INTERFACE ITF_Heatpump EXTENDS ITF_StandardFB

PROPERTY HeatpumpState : eHeatpumpState
GET
END_GET
END_PROPERTY

PROPERTY OperationMode : eHeatpumpMode
SET
END_SET
END_PROPERTY

PROPERTY Setpoint : Real
SET
END_SET
END_PROPERTY

END_INTERFACE

(* stored: Version 1.1.0.1, ProductVersion 3.1.4026.18
   Itf ITF_Heatpump: Id {81ad603a-925f-4a1a-a781-e035266bc339}
   Property HeatpumpState: Id {e84765d7-8c03-4c69-90aa-09fbaaa90fbd}
   Get Get: Id {7d37d180-4b07-4576-a3f6-55a919cc972b}
   Property OperationMode: Id {05db1adb-b4b7-42a0-b0f2-2acad7899755}
   Set Set: Id {7c757362-308e-4764-9814-e386549cc734}
   Property Setpoint: Id {3189da90-1975-4c1e-80fa-59a44dd66182}
   Set Set: Id {1548dbf7-ce76-40da-bb52-4d575df1b9b9} *)
